FUNCTION_BLOCK Test_Raises_OnSecondsChanged EXTENDS TUnitTestBase
IMPLEMENTS 
    IEventHandler_OnSecondsChanged
VAR
    NowFromEvent : TIMESTRUCT;
    
    OnSecondsChanged_Raised    : BOOL;
END_VAR

METHOD  Execute
VAR_INST
    ClockEventSource : TClockEventSource;
    Now              : TIMESTRUCT := (wDay := 23, wMonth := 12, wYear := 1945, wHour := 22, wMinute := 20, wSecond := 18);
    OneSecondLater   : TIMESTRUCT := (wDay := 23, wMonth := 12, wYear := 1945, wHour := 22, wMinute := 20, wSecond := 19);
END_VAR
OnSecondsChanged_Raised := FALSE;

ClockEventSource.Event_SecondsChanged.ClearEventHandlers().AddEventHandler(THIS^);

ClockEventSource.Init(Now := Now);
ClockEventSource(Now := OneSecondLater);

Assertion.AssertEquals_BOOL(
    Expected := TRUE,
    Actual   := OnSecondsChanged_Raised,
    ObjectName := _TestName,
    VariableName  := 'OnSecondsChanged_Raised');

Assertion.AssertEquals_STRUCT(
    Expected := OneSecondLater,
    Actual   := NowFromEvent,
    ObjectName := _TestName,
    VariableName  := 'NowFromEvent');

Test_Finished();
END_METHOD

METHOD OnSecondsChanged
VAR_INPUT
	Now	: Tc2_Utilities.TIMESTRUCT;
END_VAR
NowFromEvent := Now;
OnSecondsChanged_Raised := TRUE;
END_METHOD

END_FUNCTION_BLOCK

(* stored: Version 1.1.0.1, ProductVersion 3.1.4024.3
   POU Test_Raises_OnSecondsChanged: Id {24cee803-402d-0909-3214-8933d08be63f}, SpecialFunc None
   Method Execute: Id {cc5d5902-a3fe-0e0a-0041-841cf552b961}
   Method OnSecondsChanged: Id {07ed9024-f1fc-02c6-26de-79679bdbd9d0} *)
